Universal Robots PolyScope program: RC_E1_PLACE_130.urp

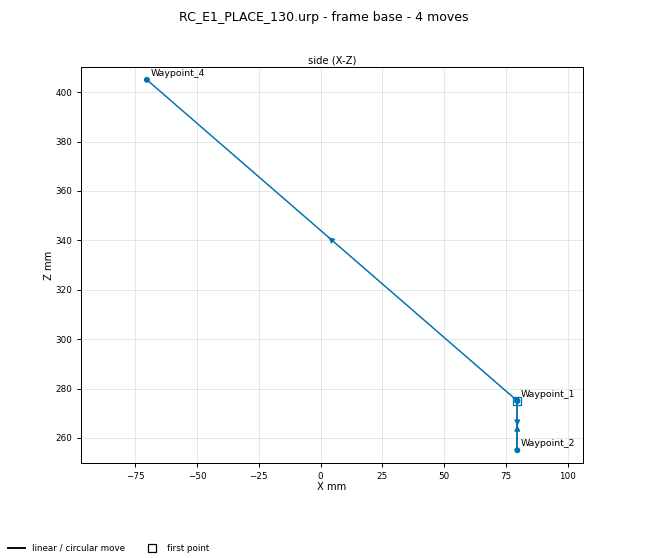
[picture p0: tool path of RC_E1_PLACE_130.urp in frame base, 4 of 4 moves have a stored position in this frame; points joined in program order, loops and branches not executed]
Program RC_E1_PLACE_130 (createdIn=3.0.0 lastSavedIn=3.0.0 directory=/programs installation=default)
Robot Program (runOnlyOnce=true motionType=MoveJ speed=1.047198 acceleration=1.396263 useActiveTCP=false)
  'Program generated by RoboDK v4.1.0 for UR3e_HORNO on 27/07/2022 12:07:02'
  'Using nominal kinematics.'
  'Using Ref. Frame No Ok 03: p[-0.386000, 1.280000, -0.011500, 0.000000, 0.000000, 0.000000]'
  'Using TCP 0208-0001-0001-307-000-3 Horno: p[0.000000, 0.000000, 0.038000, 0.000000, 0.000000, 0.000000]'
  Script: set_tcp(p[0.000000, 0.000000, 0.038000, 0.000000, 0.000000, 0.000000])
  Script: movej([0.456753, -1.863152, -0.401791, -2.476113, 1.584324, 0.464205],0.60000,0.12500,0,0.0000)
  MoveL speed 100 mm/s, acceleration 120 mm/s^2 (useActiveTCP=true)
    Waypoint Waypoint_1: TCP in base x=79.651 y=1291.057 z=275 mm, rx=2.1967 ry=-2.2136 rz=-0.0343 rad; joints [17.55, -137.114, -14.462, -120.164, 90.52, 17.98] deg; flange x=80.855 y=1291.076 z=312.981 mm, rx=2.1967 ry=-2.2136 rz=-0.0343 rad
    Waypoint Waypoint_2: TCP in base x=79.651 y=1291.057 z=255 mm, rx=2.1967 ry=-2.2136 rz=-0.0343 rad; joints [17.55, -132.15, -29.63, -109.96, 90.52, 17.98] deg; flange x=80.855 y=1291.076 z=292.981 mm, rx=2.1967 ry=-2.2136 rz=-0.0343 rad
  'Detach from 0208-0001-0001-307-000-4 Horno'
  MoveL speed 500 mm/s, acceleration 900 mm/s^2 (useActiveTCP=true)
    Waypoint Waypoint_3: TCP in base x=79.651 y=1291.057 z=275 mm, rx=2.1967 ry=-2.2136 rz=-0.0343 rad; joints [17.55, -137.114, -14.462, -120.164, 90.52, 17.98] deg; flange x=80.855 y=1291.076 z=312.981 mm, rx=2.1967 ry=-2.2136 rz=-0.0343 rad
    Waypoint Waypoint_4: TCP in base x=-70.349 y=1291.057 z=405 mm, rx=2.1967 ry=-2.2136 rz=-0.0343 rad; joints [26.17, -106.751, -23.021, -141.871, 90.775, 26.597] deg; flange x=-69.145 y=1291.076 z=442.981 mm, rx=2.1967 ry=-2.2136 rz=-0.0343 rad
